FUNCTION_BLOCK IN_ENUM_CTL (* Control block for IN_ENUM *)
  (* Standard: 61499-2 *)
  (* Version 0.0, 2004-06-21, JHC, Rockwell Automation *)
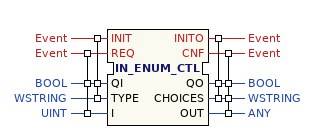
  EVENT_INPUT
    INIT WITH QI, TYPE; (* Service Initialization *)
    REQ WITH QI, I; (* Service Request *)
  END_EVENT
  EVENT_OUTPUT
    INITO WITH QO, CHOICES; (* Initialization Confirm *)
    CNF WITH QO, CHOICES, OUT; (* Confirmation of Requested Service *)
  END_EVENT
  VAR_INPUT
    QI : BOOL; (* Event Input Qualifier *)
    TYPE : WSTRING; (* Enumerated Type Name *)
    I : UINT; (* Current enumerated index *)
  END_VAR
  VAR_OUTPUT
    QO : BOOL; (* Event Output Qualifier *)
    CHOICES : WSTRING; (* Comma-separated enumeration namelist *)
    OUT : ANY; (* Enumerated variable with selected value *)
  END_VAR
END_FUNCTION_BLOCK
